FUNCTION_BLOCK FB_Observer_WORD EXTENDS FB_AbstractObserver
VAR
    _nVal:              WORD;
END_VAR

METHOD FB_init : BOOL
VAR_INPUT
	bInitRetains : BOOL; // if TRUE, the retain variables are initialized (warm start / cold start)
	bInCopyCode : BOOL;  // if TRUE, the instance afterwards gets moved into the copy code (online change)
END_VAR
THIS^._nTypeClass := __SYSTEM.TYPE_CLASS.TYPE_WORD;
THIS^._pVal := ADR(THIS^._nVal);
THIS^._nSize := SIZEOF(THIS^._nVal);
END_METHOD

PROPERTY nValue16 : WORD
GET
nValue16 := THIS^._nVal;
END_GET
END_PROPERTY

END_FUNCTION_BLOCK

(* stored: Version 1.1.0.1, ProductVersion 3.1.4024.12
   POU FB_Observer_WORD: Id {8e2c1545-b0d6-069a-20d5-19b18f4b50ad}, SpecialFunc None
   Method FB_init: Id {3ea58629-fc66-0a50-291f-d6d848673536}
   Property nValue16: Id {d4751918-9d2c-094a-235a-e569f1e92aeb}
   Get Get: Id {c8942790-c204-08ac-3ae9-f556faca894e} *)
